(* IEC 61131-3 sources: io/src/Input, 10 files *)

(* ---- IBinSignal.st ---- *)
NAMESPACE Simatic.Ax.IO.Input

    /// Interface for binary signal input handling
    /// Defines the contract for reading binary input signals with edge detection and quality status
    /// Implementations provide access to signal state, rising/falling edges, and validity information
    INTERFACE IBinSignal

        /// Returns the current state of the binary signal
        /// RETURN: TRUE if signal is active, FALSE if signal is inactive
        METHOD Q : BOOL
        END_METHOD

        /// Returns TRUE if a rising edge was detected in the current cycle
        /// Rising edge: transition from FALSE to TRUE
        /// RETURN: TRUE for one cycle after rising edge, otherwise FALSE
        METHOD QRis : BOOL
        END_METHOD

        /// Returns TRUE if a falling edge was detected in the current cycle
        /// Falling edge: transition from TRUE to FALSE
        /// RETURN: TRUE for one cycle after falling edge, otherwise FALSE
        METHOD QFal : BOOL
        END_METHOD

        /// Returns the quality status of the signal
        /// RETURN: TRUE if signal is invalid/bad, FALSE if signal is valid/good
        METHOD QBad : BOOL
        END_METHOD
    END_INTERFACE

    /// Null Object pattern implementation for ItfBinSignal
    /// Provides a safe default implementation that returns FALSE for all methods
    /// Use this to avoid null pointer checks when a binary signal is optional
    CLASS NullBinSignal
        IMPLEMENTS IBinSignal

        /// Returns the current state (always FALSE for null object)
        /// RETURN: FALSE
        METHOD PUBLIC Q : BOOL
            ;
        END_METHOD

        /// Returns rising edge status (always FALSE for null object)
        /// RETURN: FALSE
        METHOD PUBLIC QRis : BOOL
            ;
        END_METHOD

        /// Returns falling edge status (always FALSE for null object)
        /// RETURN: FALSE
        METHOD PUBLIC QFal : BOOL
            ;
        END_METHOD

        /// Returns quality status (always FALSE for null object, indicating "good" quality)
        /// RETURN: FALSE
        METHOD PUBLIC QBad : BOOL
            ;
        END_METHOD
    END_CLASS

END_NAMESPACE

(* ---- ItfBinSignal.st ---- *)
NAMESPACE Simatic.Ax.IO.Input

    /// Interface for binary signal input handling
    /// Defines the contract for reading binary input signals with edge detection and quality status
    /// Implementations provide access to signal state, rising/falling edges, and validity information
    INTERFACE ItfBinSignal

        /// Returns the current state of the binary signal
        /// RETURN: TRUE if signal is active, FALSE if signal is inactive
        METHOD Q : BOOL
        END_METHOD

        /// Returns TRUE if a rising edge was detected in the current cycle
        /// Rising edge: transition from FALSE to TRUE
        /// RETURN: TRUE for one cycle after rising edge, otherwise FALSE
        METHOD QRis : BOOL
        END_METHOD

        /// Returns TRUE if a falling edge was detected in the current cycle
        /// Falling edge: transition from TRUE to FALSE
        /// RETURN: TRUE for one cycle after falling edge, otherwise FALSE
        METHOD QFal : BOOL
        END_METHOD

        /// Returns the quality status of the signal
        /// RETURN: TRUE if signal is invalid/bad, FALSE if signal is valid/good
        METHOD QBad : BOOL
        END_METHOD
    END_INTERFACE

    /// Null Object pattern implementation for ItfBinSignal
    /// Provides a safe default implementation that returns FALSE for all methods
    /// Use this to avoid null pointer checks when a binary signal is optional
    CLASS NullBinSignal
        IMPLEMENTS ItfBinSignal

        /// Returns the current state (always FALSE for null object)
        /// RETURN: FALSE
        METHOD PUBLIC Q : BOOL
            ;
        END_METHOD

        /// Returns rising edge status (always FALSE for null object)
        /// RETURN: FALSE
        METHOD PUBLIC QRis : BOOL
            ;
        END_METHOD

        /// Returns falling edge status (always FALSE for null object)
        /// RETURN: FALSE
        METHOD PUBLIC QFal : BOOL
            ;
        END_METHOD

        /// Returns quality status (always FALSE for null object, indicating "good" quality)
        /// RETURN: FALSE
        METHOD PUBLIC QBad : BOOL
            ;
        END_METHOD
    END_CLASS

END_NAMESPACE

(* ---- BinSignal.st ---- *)
NAMESPACE Simatic.Ax.IO.Input

    /// Binary signal input handler with edge detection and inversion support
    /// Provides reading of digital input signals with automatic edge detection (rising/falling)
    /// Supports signal inversion and quality status monitoring
    /// Must be called cyclically via ReadCyclic() method
    CLASS BinSignal EXTENDS InputBase IMPLEMENTS IBinSignal
        VAR PUBLIC
            invert : BOOL := FALSE; // When TRUE, inverts the input signal (TRUE becomes FALSE and vice versa)
        END_VAR
        VAR PRIVATE
            _signalInOld : BOOL; // Previous signal state for edge detection
        END_VAR
        VAR PROTECTED
            _signalInPrefiltered : BOOL; // Signal after inversion is applied
            _statusQ : BOOL; // Current signal state
            _statusQRis : BOOL; // TRUE for one cycle when rising edge detected
            _statusQFal : BOOL; // TRUE for one cycle when falling edge detected
        END_VAR

        /// Read the binary input signal cyclically
        /// Must be called every cycle (recommended: at the beginning of the cycle)
        /// Handles signal inversion, edge detection, and quality status
        /// signal: The boolean input value from the hardware input
        /// valid: TRUE if the input is valid (periphery OK), FALSE if there's a hardware error
        /// default: Default value to use when valid = FALSE (default: FALSE)
        METHOD PUBLIC ReadCyclic
            VAR_INPUT
                signal : BOOL;
                valid : BOOL := TRUE;
                default : BOOL := FALSE;
            END_VAR

            // Apply inversion if configured and set quality status
            IF (valid) THEN
                _signalInPrefiltered :=  signal XOR invert;
                THIS.QBad(value := FALSE);
            ELSE
                _signalInPrefiltered := default;
                THIS.QBad(value := TRUE);
            END_IF;

            // Update current status and detect changes
            _statusQ := _signalInPrefiltered;
            _hasChanged := _signalInOld <> _signalInPrefiltered;

            // Detect edges: rising (FALSE->TRUE) and falling (TRUE->FALSE)
            _statusQRis := _statusQ AND NOT(_signalInOld);
            _statusQFal := NOT(_statusQ) AND _signalInOld;

            // Store current state for next cycle's edge detection
            _signalInOld := _statusQ;
        END_METHOD

        /// Returns whether the signal inversion is active
        /// RETURN: TRUE if signal is inverted, FALSE if signal is not inverted
        METHOD PUBLIC IsInverted : BOOL
            IsInverted := invert;
        END_METHOD

        /// Returns the current state of the binary signal
        /// Takes into account inversion setting and quality status
        /// RETURN: TRUE if signal is active, FALSE if signal is inactive
        METHOD PUBLIC Q : BOOL
            Q := _statusQ;
        END_METHOD

        /// Returns TRUE if a rising edge was detected in the current cycle
        /// Rising edge: transition from FALSE to TRUE (after inversion is applied)
        /// RETURN: TRUE for one cycle after rising edge, otherwise FALSE
        METHOD PUBLIC QRis : BOOL
            QRis := _statusQRis;
        END_METHOD

        /// Returns TRUE if a falling edge was detected in the current cycle
        /// Falling edge: transition from TRUE to FALSE (after inversion is applied)
        /// RETURN: TRUE for one cycle after falling edge, otherwise FALSE
        METHOD PUBLIC QFal : BOOL
            QFal := _statusQFal;
        END_METHOD
    END_CLASS
END_NAMESPACE

(* ---- BinSignalExt.st ---- *)
USING System.Timer;
NAMESPACE Simatic.Ax.IO.Input

    /// Extended binary signal input handler with configurable on-delay and off-delay timing
    /// Extends BinSignal with time-based filtering to debounce or delay signal transitions
    /// - ondelay: Delays the rising edge (FALSE->TRUE transition)
    /// - offdelay: Delays the falling edge (TRUE->FALSE transition)
    /// Useful for filtering noisy signals or implementing time-based logic
    CLASS BinSignalExt EXTENDS BinSignal
        VAR PUBLIC
            ondelay : TIME; // Delay time for rising edge (FALSE->TRUE), T#0ms = no delay
            offdelay : TIME; // Delay time for falling edge (TRUE->FALSE), T#0ms = no delay
        END_VAR
        VAR PRIVATE
            _ton : OnDelay; // Timer for on-delay functionality
            _toff : OffDelay; // Timer for off-delay functionality
            _signalInOld : BOOL; // Previous signal state for edge detection after delays
        END_VAR

        /// Read digital signal with time-based filtering
        /// Must be executed in every cycle (recommendation: beginning of cycle for digital inputs)
        /// Applies on-delay and off-delay timing to filter signal transitions
        /// signal: Digital/Boolean signal from hardware input
        /// valid: TRUE if signal is valid (periphery OK), FALSE if there's a hardware error
        /// default: Default value to use when valid = FALSE (default: FALSE)
        METHOD PUBLIC OVERRIDE ReadCyclic
            VAR_INPUT
                signal : BOOL;
                valid : BOOL := TRUE;
                default : BOOL := FALSE;
            END_VAR
            VAR_TEMP
                _tonDelayed : BOOL; // Signal after on-delay is applied
                _toffDelayed : BOOL; // Signal after off-delay is applied
            END_VAR

            // Call base class to handle inversion and quality status
            SUPER.ReadCyclic(signal := signal, valid := valid, default := default);

            // Apply on-delay: delays rising edge (FALSE->TRUE)
            IF (ondelay > T#0ms) THEN
                _ton(duration := ondelay, signal := _signalInPrefiltered);
                _tonDelayed := _ton.output;
            ELSE
                _tonDelayed := _signalInPrefiltered;
            END_IF;

            // Apply off-delay: delays falling edge (TRUE->FALSE)
            IF (offdelay > T#0ms) THEN
                _toff(duration := offdelay, signal := _signalInPrefiltered);
                _toffDelayed := _toff.output;
            ELSE
                _toffDelayed := _tonDelayed;
            END_IF;

            // Combine delayed signals: signal is TRUE if either timer is active
            _statusQ := _tonDelayed OR _toffDelayed;

            // Detect edges after delays are applied
            _statusQRis := _statusQ AND NOT(_signalInOld);
            _statusQFal := NOT(_statusQ) AND _signalInOld;
            _signalInOld := _statusQ;
        END_METHOD

    END_CLASS
END_NAMESPACE

(* ---- DintInput.st ---- *)
USING System.Math;

NAMESPACE Simatic.Ax.IO.Input

    /// Double Integer (DINT) input signal handler with quality monitoring and change detection
    /// Handles 32-bit signed integer input values from hardware or software sources
    /// Range: -2,147,483,648 to 2,147,483,647
    /// Provides tolerance-based change detection to filter minor fluctuations
    CLASS DintInput EXTENDS InputBase

        VAR PRIVATE
            _value : DINT := DINT#0; // Current input value
            _default : DINT := DINT#0; // Default value used when signal is invalid
            _qBad : BOOL; // Quality status (unused, inherited from base class)
        END_VAR

        /// Data type limits for DINT
        VAR CONSTANT PUBLIC
            MIN : DINT := DINT#-2147483648; // Minimum value for DINT data type
            MAX : DINT := DINT#2147483647; // Maximum value for DINT data type
        END_VAR

        /// Read the double integer input value cyclically
        /// Must be called every cycle to update the input value and quality status
        /// Change detection uses tolerance to avoid triggering on minor fluctuations
        /// value: The DINT input value from hardware or software source
        /// valid: TRUE if the input is valid (periphery OK), FALSE if there's a hardware error
        /// default: Default value to use when valid = FALSE (default: DINT#0)
        /// tolerance: Minimum change required to set HasChanged flag (default: DINT#0)
        METHOD PUBLIC ReadCyclic
            VAR_INPUT
                value : DINT;
                valid : BOOL := TRUE;
                default : DINT := DINT#0;
                tolerance : DINT := DINT#0;
            END_VAR

            THIS.QBad(value := NOT(valid));
            _hasChanged := ABS(_value - value) > tolerance;
            _value := value;
            _default := default;
        END_METHOD

        /// Returns the current double integer value
        /// If signal quality is good (QBad = FALSE), returns the actual value
        /// If signal quality is bad (QBad = TRUE), returns the default value
        /// RETURN: Current DINT value or default value if invalid
        METHOD PUBLIC Q : DINT
            IF (NOT(THIS.QBad())) THEN
                Q := _value;
            ELSE
                Q := _default;
            END_IF;
        END_METHOD

    END_CLASS
END_NAMESPACE

(* ---- InputBase.st ---- *)
NAMESPACE Simatic.Ax.IO.Input

    /// Base class for all input signal types
    /// Provides common functionality for quality status (QBad) and change detection
    /// This class should be extended by specific input type implementations
    CLASS InputBase
        VAR PROTECTED
            _isQBad : BOOL; // TRUE: signal is invalid (e.g., periphery error)
            _hasChanged : BOOL; // TRUE: value changed between consecutive reads
        END_VAR

        /// Set the QBad status internally
        /// Used by derived classes to indicate signal validity
        /// value: TRUE if signal is bad/invalid, FALSE if signal is good/valid
        METHOD PROTECTED QBad
            VAR_INPUT
                value : BOOL;
            END_VAR
            _isQBad := value;
        END_METHOD

        /// Returns the QBad status of the input signal
        /// QBad = TRUE indicates the signal is invalid (e.g., when valid parameter in ReadCyclic is FALSE)
        /// QBad = FALSE indicates the signal is valid and can be trusted
        /// RETURN: TRUE if signal is bad/invalid, FALSE if signal is good/valid
        METHOD PUBLIC QBad : BOOL
            QBad := _isQBad;
            ;
        END_METHOD

        /// Returns TRUE if the input value has changed between the current and previous read cycle
        /// Change detection is implemented by derived classes based on their specific data types
        /// RETURN: TRUE if value changed, FALSE if value remained the same
        METHOD PUBLIC HasChanged : BOOL;
            HasChanged := _hasChanged;
        END_METHOD

    END_CLASS
END_NAMESPACE

(* ---- IntInput.st ---- *)
USING System.Math;

NAMESPACE Simatic.Ax.IO.Input

    /// Integer (INT) input signal handler with quality monitoring and change detection
    /// Handles 16-bit signed integer input values from hardware or software sources
    /// Range: -32768 to 32767
    /// Provides tolerance-based change detection to filter minor fluctuations
    CLASS IntInput EXTENDS InputBase

        VAR PRIVATE
            _value : INT := 0; // Current input value
            _default : INT := 0; // Default value used when signal is invalid
        END_VAR

        /// Data type limits for INT
        VAR CONSTANT PUBLIC
            MAX : INT := 32767; // Maximum value for INT data type
            MIN : INT := -32768; // Minimum value for INT data type
        END_VAR

        /// Read the integer input value cyclically
        /// Must be called every cycle to update the input value and quality status
        /// Change detection uses tolerance to avoid triggering on minor fluctuations
        /// value: The INT input value from hardware or software source
        /// valid: TRUE if the input is valid (periphery OK), FALSE if there's a hardware error
        /// default: Default value to use when valid = FALSE (default: 0)
        /// tolerance: Minimum change required to set HasChanged flag (default: 0)
        METHOD PUBLIC ReadCyclic
            VAR_INPUT
                value : INT;
                valid : BOOL := TRUE;
                default : INT := 0;
                tolerance : INT := 0;
            END_VAR

            THIS.QBad(value := NOT(valid));
            _hasChanged := ABS(_value - value) > tolerance;
            _value := value;
            _default := default;
        END_METHOD

        /// Returns the current integer value
        /// If signal quality is good (QBad = FALSE), returns the actual value
        /// If signal quality is bad (QBad = TRUE), returns the default value
        /// RETURN: Current INT value or default value if invalid
        METHOD PUBLIC Q : Int
            IF (NOT(THIS.QBad())) THEN
                Q := _value;
            ELSE
                Q := _default;
            END_IF;
        END_METHOD

    END_CLASS
END_NAMESPACE

(* ---- LRealInput.st ---- *)
USING System.Math;

NAMESPACE Simatic.Ax.IO.Input

    /// Long Real (LREAL) floating-point input signal handler with quality monitoring and change detection
    /// Handles 64-bit double precision floating-point input values from hardware or software sources
    /// Range: approximately ±1.8e308 (double precision IEEE 754)
    /// Provides tolerance-based change detection to filter minor fluctuations
    /// Supports reading from LWORD (hardware format) or LREAL (software format)
    CLASS LRealInput EXTENDS InputBase

        VAR PRIVATE
            _value : LREAL := LREAL#0.0; // Current input value
            _default : LREAL := LREAL#0.0; // Default value used when signal is invalid
        END_VAR

        /// Data type limits for LREAL
        VAR CONSTANT PUBLIC
            MAX : LREAL := LREAL#1.79769313486231e+308; // Maximum positive value for LREAL data type
            MIN : LREAL := LREAL#-1.79769313486231e+308; // Maximum negative value for LREAL data type
        END_VAR

        /// Read the long real input value from hardware (LWORD format) cyclically
        /// Must be called every cycle to update the input value and quality status
        /// Converts LWORD bit pattern to LREAL floating-point value
        /// Change detection uses tolerance to avoid triggering on minor fluctuations
        /// value: The LWORD input value from hardware (bit pattern representing LREAL)
        /// valid: TRUE if the input is valid (periphery OK), FALSE if there's a hardware error
        /// default: Default value to use when valid = FALSE (default: LREAL#0.0)
        /// tolerance: Minimum change required to set HasChanged flag (default: LREAL#0.0)
        METHOD PUBLIC ReadCyclic
            VAR_INPUT
                value : LWORD;
                valid : BOOL := TRUE;
                default : LREAL := LREAL#0.0;
                tolerance : LREAL := LREAL#0.0;
            END_VAR

            THIS.QBad(value := NOT(valid));
            _hasChanged := ABS(_value - TO_LREAL(value)) > tolerance;
            _value := TO_LREAL(value);
            _default := default;
        END_METHOD

        /// Read the long real input value from software (LREAL format) cyclically
        /// Must be called every cycle to update the input value and quality status
        /// Change detection uses tolerance to avoid triggering on minor fluctuations
        /// value: The LREAL input value from software source
        /// valid: TRUE if the input is valid, FALSE if there's an error
        /// default: Default value to use when valid = FALSE (default: LREAL#0.0)
        /// tolerance: Minimum change required to set HasChanged flag (default: LREAL#0.0)
        METHOD PUBLIC ReadCyclic
            VAR_INPUT
                value : LREAL;
                valid : BOOL := TRUE;
                default : LREAL := LREAL#0.0;
                tolerance : LREAL := LREAL#0.0;
            END_VAR

            THIS.QBad(value := NOT(valid));
            _hasChanged := ABS(_value - value) > tolerance;
            _value := value;
            _default := default;
        END_METHOD

        /// Returns the current long real floating-point value
        /// If signal quality is good (QBad = FALSE), returns the actual value
        /// If signal quality is bad (QBad = TRUE), returns the default value
        /// RETURN: Current LREAL value or default value if invalid
        METHOD PUBLIC Q : LREAL
            IF (NOT(THIS.QBad())) THEN
                Q := _value;
            ELSE
                Q := _default;
            END_IF;
        END_METHOD

    END_CLASS
END_NAMESPACE

(* ---- RealInput.st ---- *)
USING System.Math;

NAMESPACE Simatic.Ax.IO.Input

    /// Real (REAL) floating-point input signal handler with quality monitoring and change detection
    /// Handles 32-bit floating-point input values from hardware or software sources
    /// Range: approximately ±3.4e38 (single precision IEEE 754)
    /// Provides tolerance-based change detection to filter minor fluctuations
    /// Supports reading from DWORD (hardware format) or REAL (software format)
    CLASS RealInput EXTENDS InputBase

        VAR PRIVATE
            _value : REAL := REAL#0.0; // Current input value
            _default : REAL := REAL#0.0; // Default value used when signal is invalid
        END_VAR

        /// Data type limits for REAL
        VAR CONSTANT PUBLIC
            MAX : REAL := REAL#+3.402823e+38; // Maximum positive value for REAL data type
            MIN : REAL := REAL#-3.402823e+38; // Maximum negative value for REAL data type
        END_VAR

        /// Read the real input value from hardware (DWORD format) cyclically
        /// Must be called every cycle to update the input value and quality status
        /// Converts DWORD bit pattern to REAL floating-point value
        /// Change detection uses tolerance to avoid triggering on minor fluctuations
        /// value: The DWORD input value from hardware (bit pattern representing REAL)
        /// valid: TRUE if the input is valid (periphery OK), FALSE if there's a hardware error
        /// default: Default value to use when valid = FALSE (default: REAL#0.0)
        /// tolerance: Minimum change required to set HasChanged flag (default: REAL#0.0)
        METHOD PUBLIC ReadCyclic
            VAR_INPUT
                value : DWORD;
                valid : BOOL := TRUE;
                default : REAL := REAL#0.0;
                tolerance : REAL := REAL#0.0;
            END_VAR

            THIS.QBad(value := NOT(valid));
            _hasChanged := ABS(_value - TO_REAL(value)) > tolerance;
            _value := TO_REAL(value);
            _default := default;
        END_METHOD

        /// Read the real input value from software (REAL format) cyclically
        /// Must be called every cycle to update the input value and quality status
        /// Change detection uses tolerance to avoid triggering on minor fluctuations
        /// value: The REAL input value from software source
        /// valid: TRUE if the input is valid, FALSE if there's an error
        /// default: Default value to use when valid = FALSE (default: REAL#0.0)
        /// tolerance: Minimum change required to set HasChanged flag (default: REAL#0.0)
        METHOD PUBLIC ReadCyclic
            VAR_INPUT
                value : REAL;
                valid : BOOL := TRUE;
                default : REAL := REAL#0.0;
                tolerance : REAL := REAL#0.0;
            END_VAR

            THIS.QBad(value := NOT(valid));
            _hasChanged := ABS(_value - value) > tolerance;
            _value := value;
            _default := default;
        END_METHOD

        /// Returns the current real floating-point value
        /// If signal quality is good (QBad = FALSE), returns the actual value
        /// If signal quality is bad (QBad = TRUE), returns the default value
        /// RETURN: Current REAL value or default value if invalid
        METHOD PUBLIC Q : REAL
            IF (NOT(THIS.QBad())) THEN
                Q := _value;
            ELSE
                Q := _default;
            END_IF;
        END_METHOD

    END_CLASS
END_NAMESPACE

(* ---- WordInput.st ---- *)
NAMESPACE Simatic.Ax.IO.Input

    /// Word (WORD) input signal handler with quality monitoring and change detection
    /// Handles 16-bit unsigned word input values from hardware or software sources
    /// Range: 0 (16#0) to 65535 (16#FFFF)
    /// Typically used for bit patterns, status words, or unsigned integer values
    CLASS WordInput EXTENDS InputBase

        VAR PRIVATE
            _value : WORD := WORD#16#0; // Current input value
            _default : WORD := WORD#16#0; // Default value used when signal is invalid
        END_VAR

        /// Data type limits for WORD
        VAR CONSTANT PUBLIC
            MIN : WORD := WORD#16#0; // Minimum value for WORD data type (0)
            MAX : WORD := WORD#16#FFFF; // Maximum value for WORD data type (65535)
        END_VAR

        /// Read the word input value cyclically
        /// Must be called every cycle to update the input value and quality status
        /// Change detection triggers on any bit change
        /// value: The WORD input value from hardware or software source
        /// valid: TRUE if the input is valid (periphery OK), FALSE if there's a hardware error
        /// default: Default value to use when valid = FALSE (default: WORD#16#0)
        METHOD PUBLIC ReadCyclic
            VAR_INPUT
                value : WORD;
                valid : BOOL := TRUE;
                default : WORD := WORD#16#0;
            END_VAR

            THIS.QBad(value := NOT(valid));
            _hasChanged := _value <> value;
            _value := value;
            _default := default;
        END_METHOD

        /// Returns the current word value
        /// If signal quality is good (QBad = FALSE), returns the actual value
        /// If signal quality is bad (QBad = TRUE), returns the default value
        /// RETURN: Current WORD value or default value if invalid
        METHOD PUBLIC Q : WORD
            IF (NOT(THIS.QBad())) THEN
                Q := _value;
            ELSE
                Q := _default;
            END_IF;
        END_METHOD

    END_CLASS
END_NAMESPACE
